FUNCTION_BLOCK AD_AND_4 (* FB to calculate bitwise AND (generic FB) Adapter-Ausgang wird nur bei Wertänderung aktualisiert (Event nur bei tatsächlicher Änderung). *)
  (* Standard: 61499-2; Description: Copyright (c) 2026 HR Agrartechnik GmbH This program and the accompanying materials are made available under the terms of the Eclipse Public License 2.0 which is available at https://www.eclipse.org/legal/epl-2.0/ SPDX-License-Identifier: EPL-2.0 *)
  (* Version 1.0, 2026-08-13, Franz Höpfinger, HR Agrartechnik GmbH, initial API and implementation and/or initial documentation *)
  PACKAGE adapter::bitwiseOperators;
  IMPORT eclipse4diac::core::GenericClassName;
  {SET_ATTRIBUTE(eclipse4diac::core::GenericClassName, 'GEN_AD_AND')}
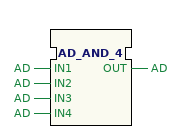
  SOCKETS
    IN1 : adapter::types::unidirectional::AD; (* AND input 1 *)
    IN2 : adapter::types::unidirectional::AD; (* AND input 2 *)
    IN3 : adapter::types::unidirectional::AD; (* AND input 3 *)
    IN4 : adapter::types::unidirectional::AD; (* AND input 4 *)
  END_SOCKETS
  PLUGS
    OUT : adapter::types::unidirectional::AD; (* AND result *)
  END_PLUGS
END_FUNCTION_BLOCK
